{attribute 'GeneratedUsingTerminal: EL3773-0000-0016'}
{attribute addProperty BoxType "EL3773-0000-0016"}
{attribute addProperty Id "U1_STATUSAT %I*U1_STATUS_B07533568"}
{attribute addProperty CRC "2018444205"}
{attribute addProperty Size "8"}
TYPE L1_Voltage_Status_784F03AD EXTENDS InputBase_8311D824 :
STRUCT
	{attribute addProperty Name "U1_STATUS"}
	U1_STATUS AT %I* : U1_STATUS_B0753356;
END_STRUCT
END_TYPE

(* stored: Version 1.2.0.0, ProductVersion 3.1.4024.9
   DUT L1_Voltage_Status_784F03AD: Id {8d529aa3-6cab-4f55-bf86-de3c55087384} *)
